// Type alias for a wide string with a maximum length of 255 characters.
TYPE T_MaxWString : WSTRING(255); END_TYPE

(* stored: Version 1.1.0.1
   DUT T_MaxWString: Id {0760c1fa-a817-0d86-0f0c-9a2e5d271a39} *)
